Universal Robots PolyScope program: chinf_demo.urp

Program chinf_demo (installation=default directory=/programs/usbdisk_2 createdIn=3.8.0.61336 lastSavedIn=3.9.0.64176 robotSerialNumber=2015330452)
Calibrated DH parameters: a=[0.000022, -0.243108, -0.198419, 0.000083, 0.000037, 0]; d=[0.152032, 7.022349, 13.600006, -20.509484, 0.085332, 0.082316]; alpha=[1.57032, -0.003617, -0.003833, 1.570553, -1.570903, 0]; deltaTheta=[-0.000133, -0.104117, -0.274955, 0.379047, -0.000031, 0.000084]
BeforeStart
  URCap Gripper Activate (Robotiq_Grippers, Robotiq Inc.) dataModel(ResetAndActivateKey=false)
  Script file /programs/usbdisk_2/CHINF.script
    | def poseMoveHandler(pose,action):
    |     movej(pose)
    |     socket_send_string(action)
    | end
    | 
    | def getServerActionAndPose():
    |     global receiveAction=socket_read_string()
    |     socket_send_string(receiveAction)
    | 
    |     global receivePose=socket_read_ascii_float(6)
    |     while (receivePose[0] !=6):
    |         global receivePose=socket_read_ascii_float(6)
    |     end
    |     socket_send_string(receivePose)
    | end
    | 
    | def floatToPose(receiveFromServ):
    |     global targetPos=p[0,0,0,0,0,0]
    |     global counter=0
    |     while (counter < 6):
    |         targetPos[counter]=receiveFromServ[counter+1]
    |         global counter=counter+1
    |     end
    |     return targetPos
    | end
    | def floatToJoint(receiveFromServ):
    |     global targetPos=[0,0,0,0,0,0]
    |     global counter=0
    |     while (counter < 6):
    |         targetPos[counter]=receiveFromServ[counter+1]
    |         global counter=counter+1
    |     end
    |     return targetPos
    | end
    | 
    | def sendPoseWithCMD():
    |     freedrive_mode()
    |     socket_send_string("freedrive_mode")
    | 
    |     global stausCode = socket_read_byte_list(1)
    |     while (stausCode[0] != 1):
    |         global stausCode = socket_read_byte_list(1)
    |     end
    | 
    |     global isFreeDrive = (stausCode[1] == 2)
    |     if (isFreeDrive):
    |         global endCode = socket_read_byte_list(1)
    |         while (endCode[0] != 1):
    |             global endCode = socket_read_byte_list(1)
    |         end
    |         p = get_actual_tcp_pose()
    |         socket_send_string(p)
    |         end_freedrive_mode()
    |     end
    | end
    | 
    | def movePoseWithCMD():
    |     socket_send_string("move")
    |     receivePose=socket_read_ascii_float(6)
    |     while (receivePose[0] !=6):
    |         receivePose=socket_read_ascii_float(6)
    |     end
    |     pose = floatToPose(receivePose)
    |     movej(pose)
    | end
    | 
    | def moveJointWithCMD():
    |     socket_send_string("moveJoint")
    | 	wantGetLen = 2
    |     global MoveJoint=socket_read_ascii_float(wantGetLen)
    |     while (MoveJoint[0] !=wantGetLen):
    |         global MoveJoint=socket_read_ascii_float(wantGetLen)
    |     end
    |     pose = get_actual_joint_positions()
    |     pose[MoveJoint[1]] = pose[MoveJoint[1]]+MoveJoint[2]
    |     servoj(pose,0,0,2)
    | end
    | 
    | def ForceMode():
    | 	socket_send_string("ForceMode")
    | 	wantGetLen = 2
    | 	 global ForceModeFloat=socket_read_ascii_float(wantGetLen)
    | 		while (ForceModeFloat[0] !=wantGetLen):
    | 			global ForceModeFloat=socket_read_ascii_float(wantGetLen)
    | 		end
    | 	global forceJointNumber = ForceModeFloat[1]
    | 	global JointForce = ForceModeFloat[2]
    | 	axis = [0, 0, 0, 0, 0, 0]
    | 	Force = [0, 0, 0, 0, 0, 0]
    | 	axis[forceJointNumber] = 1
    | 	Force[forceJointNumber] = JointForce
    | 	force_mode( tool_pose(), axis, Force, 2, [0.1, 0.1, 0.15, 0.17, 0.17, 0.17])
    | end
  open := socket_open("192.168.1.109",1100)
  Loop While (checkContinuously=false) expression=not open
    open := socket_open("192.168.1.109",1100)
Robot Program (runOnlyOnce=false)
  statusCode := socket_read_byte_list(1)
  Loop While (checkContinuously=false) expression=statusCode[0]≠1
    statusCode := socket_read_byte_list(1)
  If statusCode[1]≟1
    Script: sendPoseWithCMD()
  ElseIf statusCode[1]≟2
    Script: moveJointWithCMD()
  ElseIf statusCode[1]≟33
    URCap Gripper (Robotiq_Grippers, Robotiq Inc.) dataModel(position=0.0, force=100.0, speed=100.0, positionInDouble=0.0, forceInDouble=100.0, speedInDouble=100.0, slaveIds=[9], blocking=true)
  ElseIf statusCode[1]≟13
    URCap Gripper (Robotiq_Grippers, Robotiq Inc.) dataModel(position=100.0, force=100.0, speed=0.0, positionInDouble=100.0, forceInDouble=100.0, speedInDouble=0.0, slaveIds=[9], blocking=true)
  ElseIf statusCode[1]≟23
    URCap Gripper (Robotiq_Grippers, Robotiq Inc.) dataModel(position=100.0, force=0.0, speed=0.0, positionInDouble=100.0, forceInDouble=0.0, speedInDouble=0.0, slaveIds=[9], blocking=true)
  ElseIf statusCode[1]≟11
    Script: movePoseWithCMD()
  ElseIf statusCode[1]≟4
    Script: ForceMode()
  ElseIf statusCode[1]≟44
    Script: end_force_mode()
